// TIA Portal V16 export
// export: Created 2021-07-06T05:47:26.2051542Z, ExportSetting WithDefaults, DisplayName Totally Integrated Automation Portal, DisplayVersion V16 Update 4, DisplayName TIA Portal Version Control Interface, DisplayVersion V16 Update 2, DisplayName TIA Portal Openness, DisplayVersion V16 Update 4, DisplayName STEP 7 Professional, DisplayVersion V16 Update 4, DisplayName STEP 7 Safety, DisplayVersion V16, DisplayName WinCC Advanced, DisplayVersion V16 Update 4
FUNCTION_BLOCK "Main_Safety_RTG1"   // FB1, F_FBD
{ S7_Optimized_Access := 'TRUE' }
VERSION : 0.1
// stored: AutoNumber false, IsIECCheckEnabled false, UDAEnableTagReadback false
   VAR
      faults_clear : Bool;
      running : Bool;
   END_VAR
   VAR_TEMP
      a_ok : Bool;
      b_ok : Bool;
      clear_to_run : Bool;
   END_VAR
BEGIN

REGION Network 1
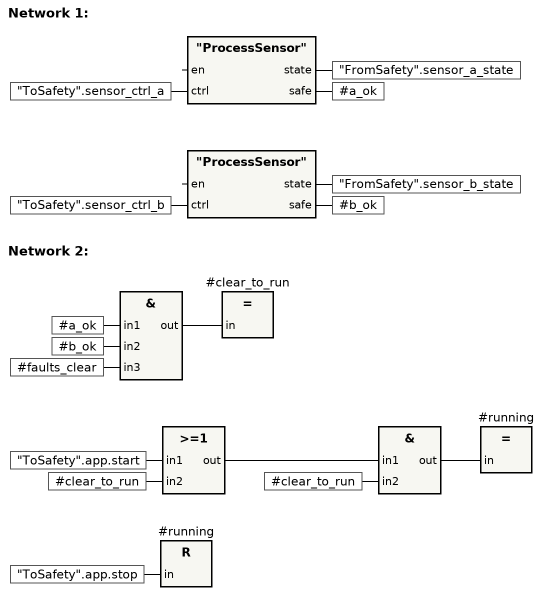
   "ProcessSensor"(ctrl := "ToSafety".sensor_ctrl_a, state => "FromSafety".sensor_a_state, safe => #a_ok);
   "ProcessSensor"(ctrl := "ToSafety".sensor_ctrl_b, state => "FromSafety".sensor_b_state, safe => #b_ok);
END_REGION

REGION Network 2
   #clear_to_run := #a_ok AND #b_ok AND #faults_clear;
   #running := ("ToSafety".app.start OR #clear_to_run) AND #clear_to_run;
   IF "ToSafety".app.stop THEN #running := FALSE; END_IF;
END_REGION
END_FUNCTION_BLOCK
